PROGRAM Main
VAR
    // Simulated motor that is always allowed to move
    {attribute 'pytmc' := '
        pv: PLC:TST:MOT:SIM:01
        field: DESC Simulated Working Motor
    '}
    M1: DUT_MotionStage;
    fbMotion1: FB_MotionStageSim;

    // Simulated motor that is never allowed to move
    {attribute 'pytmc' := '
        pv: PLC:TST:MOT:SIM:02
        field: DESC Simulated Broken Motor
    '}
    M2: DUT_MotionStage;
    fbMotion2: FB_MotionStage;

    // Simulated motor with limits at 0 and 100
    {attribute 'pytmc' := '
        pv: PLC:TST:MOT:SIM:03
        field: DESC Simulated Working Motor With Limits
    '}
    M3: DUT_MotionStage;
    fbMotion3: FB_MotionStage;

    stM1Extra : DUT_MotionStage_Extras;
    stM2Extra : DUT_MotionStage_Extras;
    stM3Extra : DUT_MotionStage_Extras;

END_VAR

fbMotion1(stMotionStage := M1);
fbMotion2(stMotionStage := M2);
fbMotion3(stMotionStage := M3);
M3.bHardwareEnable := TRUE;
M3.bPowerSelf := TRUE;
M3.bLimitForwardEnable := M3.Axis.NcToPlc.ActPos < 99.7;
M3.bLimitBackwardEnable := M3.Axis.NcToPlc.ActPos > 0.2;

(* Update extras for visualization purposes *)
stM1Extra.bVisuHighLim := NOT M1.bAllForwardEnable;
stM1Extra.bVisuLowLim := NOT M1.bAllBackwardEnable;

stM2Extra.bVisuHighLim := NOT M2.bAllForwardEnable;
stM2Extra.bVisuLowLim := NOT M2.bAllBackwardEnable;

stM3Extra.bVisuHighLim := NOT M3.bAllForwardEnable;
stM3Extra.bVisuLowLim := NOT M3.bAllBackwardEnable;

END_PROGRAM

(* stored: Version 1.1.0.1, ProductVersion 3.1.4024.4
   POU Main: Id {7b41e58a-08f0-4959-90b4-af08ef5cbf10}, SpecialFunc None *)
